// vecB=VecA*num
FUNCTION vecDot : LREAL
VAR_IN_OUT CONSTANT
	vecA :ARRAY[*] OF LREAL;
	vecB :ARRAY[*] OF LREAL;
END_VAR

VAR
	m :DINT;
	i :DINT;
END_VAR

m:=UPPER_BOUND(vecA,1);
ASSERT(UPPER_BOUND(VecB,1)=m);

vecDot :=0;
FOR i:=1 TO m DO
	vecDot := vecDot + vecA[i]*vecB[i];
END_FOR

END_FUNCTION

(* stored: Version 1.1.0.1, ProductVersion 3.1.4024.12
   POU vecDot: Id {dd510cc3-aa03-4332-b7d2-fe1b23cb1742}, SpecialFunc None *)
